// TIA Portal V16 export
// export: Created 2024-04-23T10:19:32.5105777Z, ExportSetting WithDefaults, DisplayName Totally Integrated Automation Portal, DisplayVersion V16 Update 5, DisplayName TIA Portal Version Control Interface, DisplayVersion V16 Update 2, DisplayName TIA Portal Openness, DisplayVersion V16 Update 5, DisplayName TIA Portal Teamcenter Gateway, DisplayVersion V16, DisplayName SINAMICS Startdrive Advanced, DisplayVersion V16, DisplayName SINAMICS Startdrive G130, G150, S120, S150, SINAMICS MV, S210, DisplayVersion V16, DisplayName SINAMICS Startdrive G110M, G120, G120C, G120D, G120P, DisplayVersion V16, DisplayName STEP 7 Professional, DisplayVersion V16 Update 5, DisplayName STEP 7 Safety, DisplayVersion V16, DisplayName WinCC UA Professional, DisplayVersion V16 Update 5
DATA_BLOCK "Serie de Fourier_DB"   // DB6
VERSION : 0.1
// stored: AutoNumber true, DBAccessibleFromOPCUA true, InstanceOfName Serie de Fourier, InstanceOfType FB
"Serie de Fourier"
   // VAR_INPUT
   //    "Enable Serie" : Bool;
   //    "Tm (ms)" : Real;
   //    Amplitud : Real;
   //    "Periodo (s)" : Real;
   //    N_Fourier : Int;
   // END_VAR
   // VAR_OUTPUT
   //    "Serie f(t)" : Real;
   // END_VAR
   // VAR
   //    cont { ExternalAccessible := 'False'; ExternalVisible := 'False'; ExternalWritable := 'False'} : Int;
   // END_VAR
BEGIN
END_DATA_BLOCK
